// Mitsubishi GX Developer project: lab 3   PLC: FX series

PROGRAM MAIN
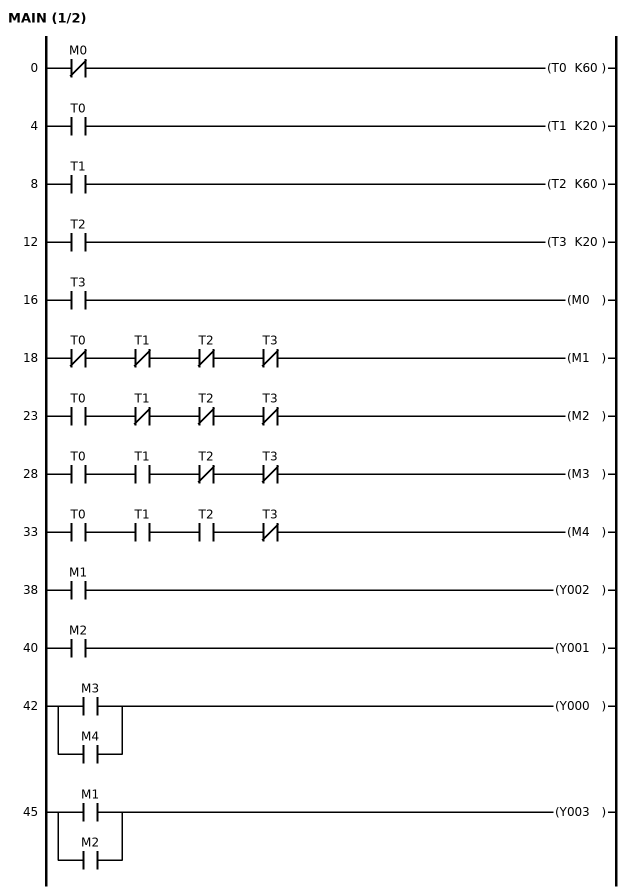
0     LDI     M0
      OUT     T0 K60
4     LD      T0
      OUT     T1 K20
8     LD      T1
      OUT     T2 K60
12    LD      T2
      OUT     T3 K20
16    LD      T3
      OUT     M0
18    LDI     T0
      ANI     T1
      ANI     T2
      ANI     T3
      OUT     M1
23    LD      T0
      ANI     T1
      ANI     T2
      ANI     T3
      OUT     M2
28    LD      T0
      AND     T1
      ANI     T2
      ANI     T3
      OUT     M3
33    LD      T0
      AND     T1
      AND     T2
      ANI     T3
      OUT     M4
38    LD      M1
      OUT     Y002
40    LD      M2
      OUT     Y001
42    LD      M3
      OR      M4
      OUT     Y000
45    LD      M1
      OR      M2
      OUT     Y003
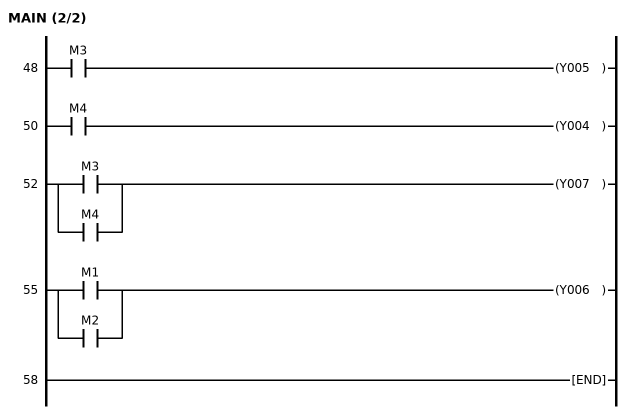
48    LD      M3
      OUT     Y005
50    LD      M4
      OUT     Y004
52    LD      M3
      OR      M4
      OUT     Y007
55    LD      M1
      OR      M2
      OUT     Y006
58    END
END_PROGRAM
